(* Logix 5000 project; controller Sucrose_Main Emulate 5570 rev 20.12; software revision 20.01; part 12 of 30 *)
(* tags used below, declared in another part *)
   AI_E21_0 : REAL[8];   // Analog Input EN2T_FLX 192.168.1.21
   AI_E21_1 : REAL[8];   // Analog Input EN2T_FLX 192.168.1.21
   AI_E21_2 : REAL[8];   // Analog Input EN2T_FLX 192.168.1.21
   HOT_WATER_FLOW : DINT;
   HOT_WATER_TEMP : DINT;
   HRM_SIP250TimeRemaining : DINT;
   HRM_SIP254TimeRemaining : DINT;
   HRM_StepTimeRemaining : DINT;
   Integrity_Control : CONTROL;
   Integrity_Result : DINT;
   Integrity_Test_FIFO : REAL[15];
   New_Sec : BOOL;
   ONESHOTBITS : INT[10];
   Rung_Comment : BOOL;
   SucroseDischarge : Area_Program;
   SucroseFiltration : Area_Program;
   temp_toggle : BOOL;
   toggle : BOOL;
(* FiltrationArea_AutoLogic, continued *)

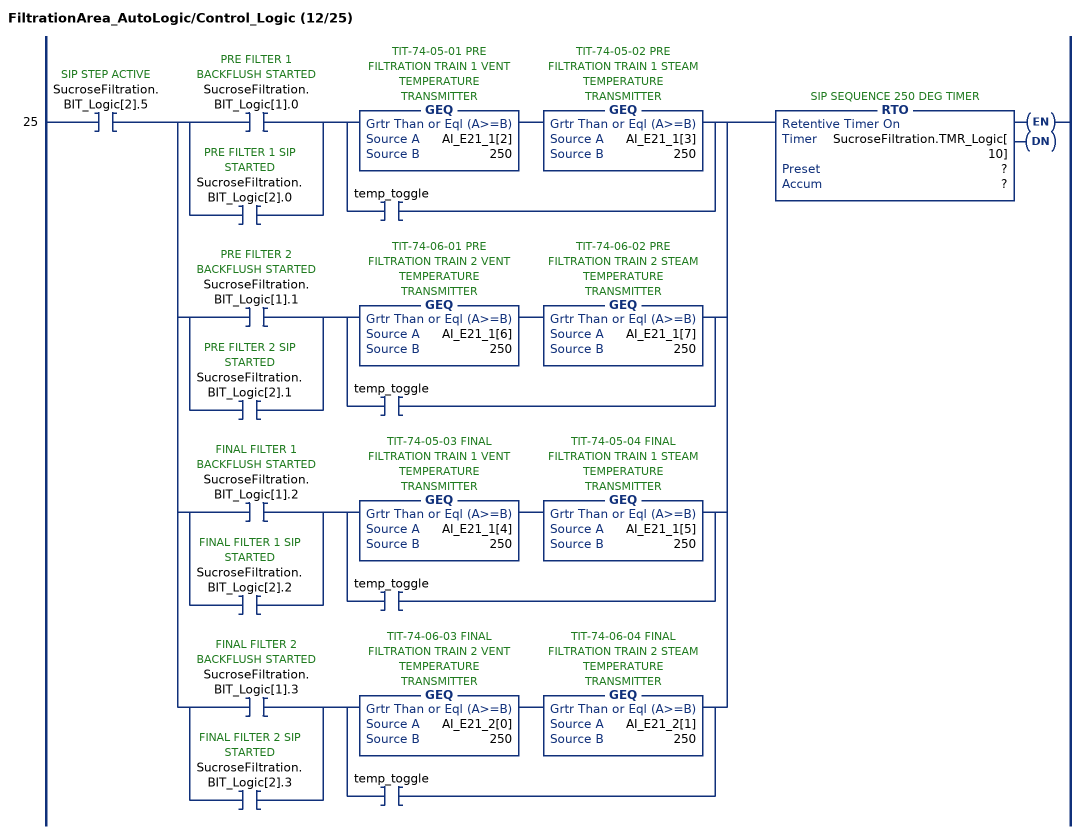
   25: XIC(SucroseFiltration.BIT_Logic[2].5)[[XIC(SucroseFiltration.BIT_Logic[1].0) ,XIC(SucroseFiltration.BIT_Logic[2].0) ] [GEQ(AI_E21_1[2],250) GEQ(AI_E21_1[3],250) ,XIC(temp_toggle) ] ,[XIC(SucroseFiltration.BIT_Logic[1].1) ,XIC(SucroseFiltration.BIT_Logic[2].1) ] [GEQ(AI_E21_1[6],250) GEQ(AI_E21_1[7],250) ,XIC(temp_toggle) ] ,[XIC(SucroseFiltration.BIT_Logic[1].2) ,XIC(SucroseFiltration.BIT_Logic[2].2) ] [GEQ(AI_E21_1[4],250) GEQ(AI_E21_1[5],250) ,XIC(temp_toggle) ] ,[XIC(SucroseFiltration.BIT_Logic[1].3) ,XIC(SucroseFiltration.BIT_Logic[2].3) ] [GEQ(AI_E21_2[0],250) GEQ(AI_E21_2[1],250) ,XIC(temp_toggle) ] ]RTO(SucroseFiltration.TMR_Logic[10],?,?);
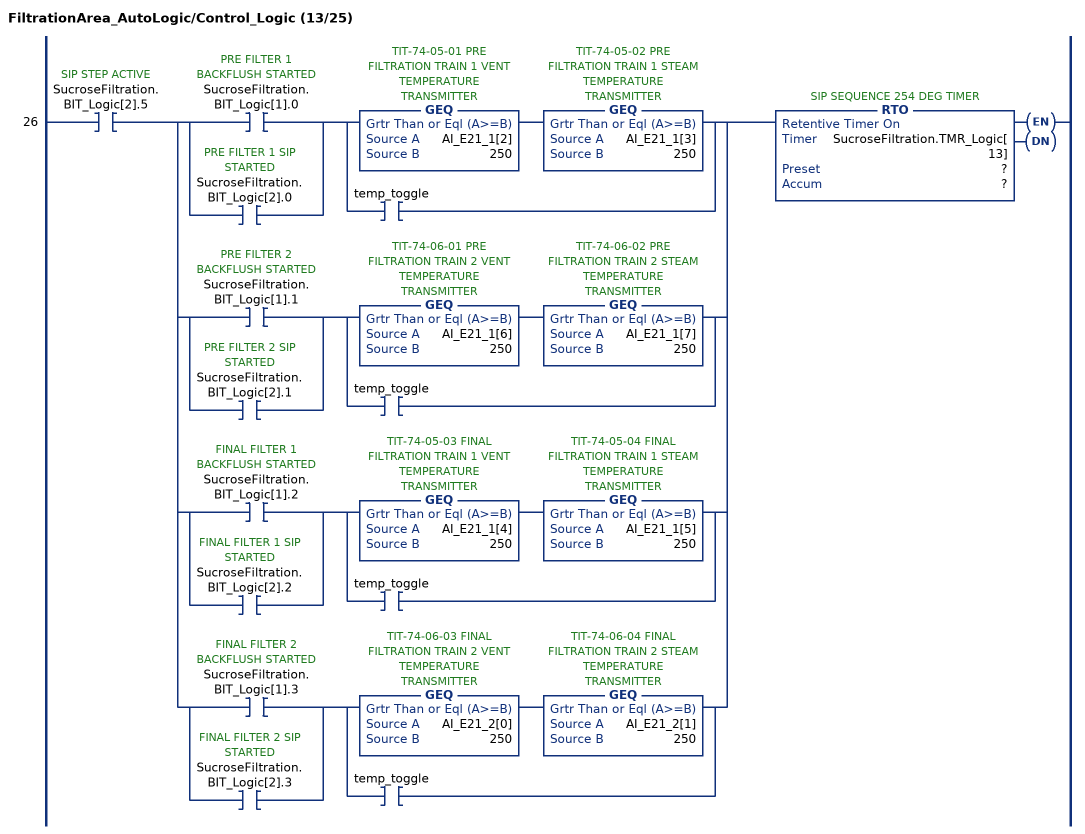
   26: XIC(SucroseFiltration.BIT_Logic[2].5)[[XIC(SucroseFiltration.BIT_Logic[1].0) ,XIC(SucroseFiltration.BIT_Logic[2].0) ] [GEQ(AI_E21_1[2],250) GEQ(AI_E21_1[3],250) ,XIC(temp_toggle) ] ,[XIC(SucroseFiltration.BIT_Logic[1].1) ,XIC(SucroseFiltration.BIT_Logic[2].1) ] [GEQ(AI_E21_1[6],250) GEQ(AI_E21_1[7],250) ,XIC(temp_toggle) ] ,[XIC(SucroseFiltration.BIT_Logic[1].2) ,XIC(SucroseFiltration.BIT_Logic[2].2) ] [GEQ(AI_E21_1[4],250) GEQ(AI_E21_1[5],250) ,XIC(temp_toggle) ] ,[XIC(SucroseFiltration.BIT_Logic[1].3) ,XIC(SucroseFiltration.BIT_Logic[2].3) ] [GEQ(AI_E21_2[0],250) GEQ(AI_E21_2[1],250) ,XIC(temp_toggle) ] ]RTO(SucroseFiltration.TMR_Logic[13],?,?);
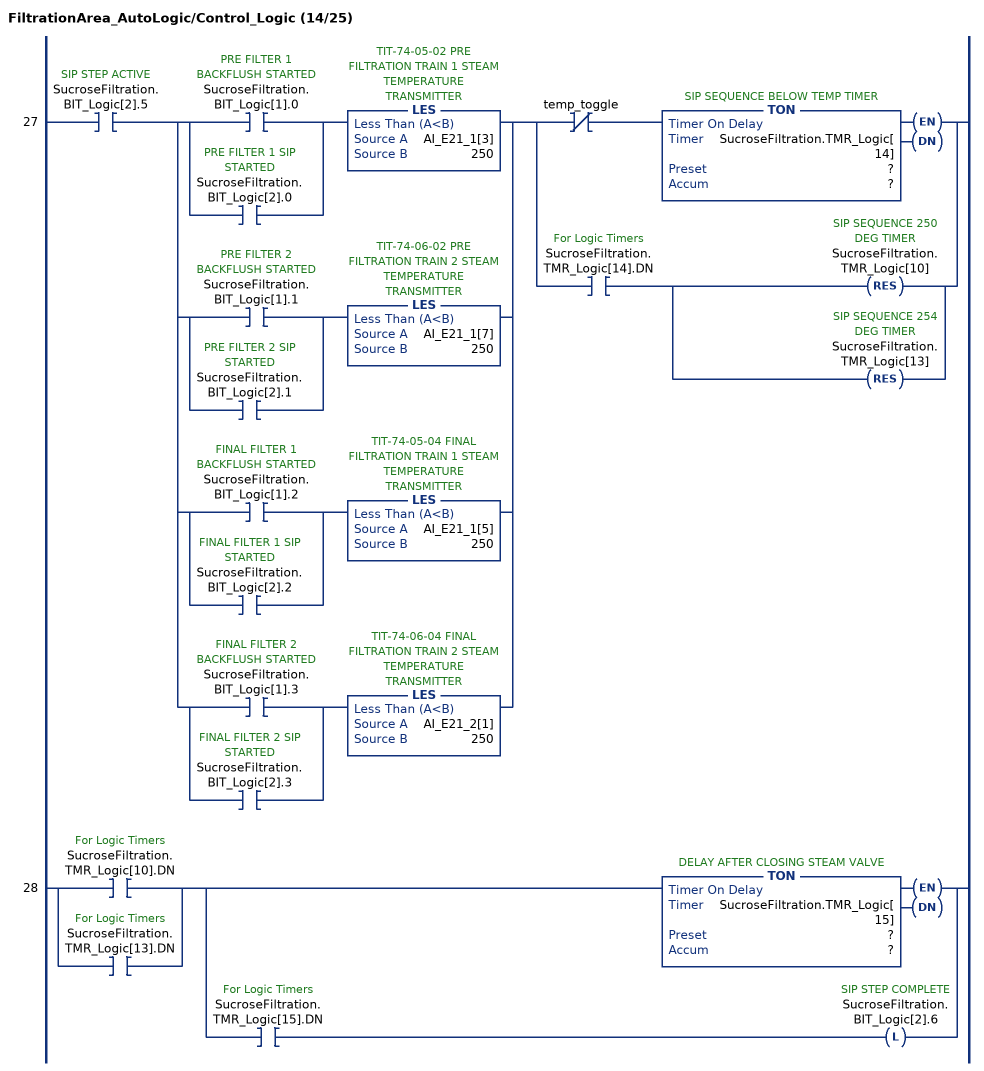
   27: XIC(SucroseFiltration.BIT_Logic[2].5)[[XIC(SucroseFiltration.BIT_Logic[1].0) ,XIC(SucroseFiltration.BIT_Logic[2].0) ] LES(AI_E21_1[3],250) ,[XIC(SucroseFiltration.BIT_Logic[1].1) ,XIC(SucroseFiltration.BIT_Logic[2].1) ] LES(AI_E21_1[7],250) ,[XIC(SucroseFiltration.BIT_Logic[1].2) ,XIC(SucroseFiltration.BIT_Logic[2].2) ] LES(AI_E21_1[5],250) ,[XIC(SucroseFiltration.BIT_Logic[1].3) ,XIC(SucroseFiltration.BIT_Logic[2].3) ] LES(AI_E21_2[1],250) ][XIO(temp_toggle) TON(SucroseFiltration.TMR_Logic[14],?,?) ,XIC(SucroseFiltration.TMR_Logic[14].DN) [RES(SucroseFiltration.TMR_Logic[10]) ,RES(SucroseFiltration.TMR_Logic[13]) ] ];
   28: [XIC(SucroseFiltration.TMR_Logic[10].DN) ,XIC(SucroseFiltration.TMR_Logic[13].DN) ][TON(SucroseFiltration.TMR_Logic[15],?,?) ,XIC(SucroseFiltration.TMR_Logic[15].DN) OTL(SucroseFiltration.BIT_Logic[2].6) ];
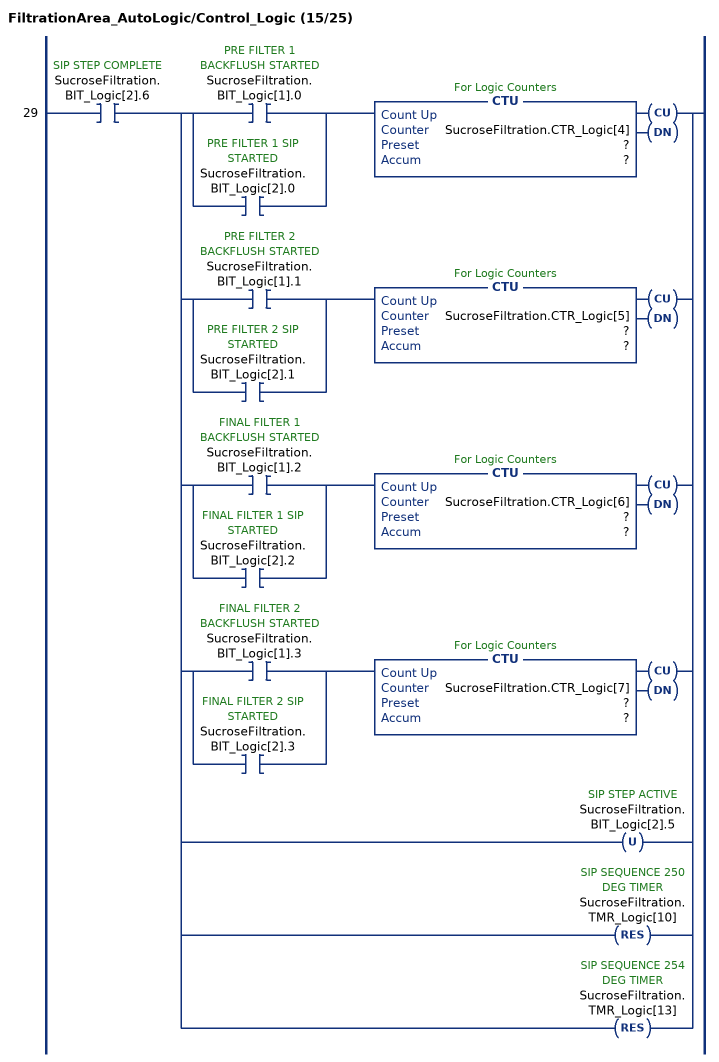
   29: XIC(SucroseFiltration.BIT_Logic[2].6)[[XIC(SucroseFiltration.BIT_Logic[1].0) ,XIC(SucroseFiltration.BIT_Logic[2].0) ] CTU(SucroseFiltration.CTR_Logic[4],?,?) ,[XIC(SucroseFiltration.BIT_Logic[1].1) ,XIC(SucroseFiltration.BIT_Logic[2].1) ] CTU(SucroseFiltration.CTR_Logic[5],?,?) ,[XIC(SucroseFiltration.BIT_Logic[1].2) ,XIC(SucroseFiltration.BIT_Logic[2].2) ] CTU(SucroseFiltration.CTR_Logic[6],?,?) ,[XIC(SucroseFiltration.BIT_Logic[1].3) ,XIC(SucroseFiltration.BIT_Logic[2].3) ] CTU(SucroseFiltration.CTR_Logic[7],?,?) ,OTU(SucroseFiltration.BIT_Logic[2].5) ,RES(SucroseFiltration.TMR_Logic[10]) ,RES(SucroseFiltration.TMR_Logic[13]) ];
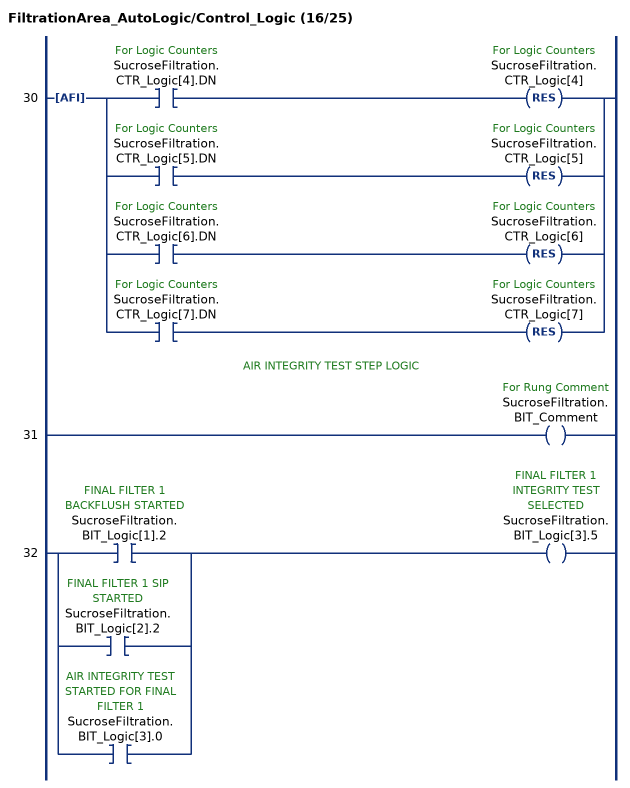
   30: AFI()[XIC(SucroseFiltration.CTR_Logic[4].DN) RES(SucroseFiltration.CTR_Logic[4]) ,XIC(SucroseFiltration.CTR_Logic[5].DN) RES(SucroseFiltration.CTR_Logic[5]) ,XIC(SucroseFiltration.CTR_Logic[6].DN) RES(SucroseFiltration.CTR_Logic[6]) ,XIC(SucroseFiltration.CTR_Logic[7].DN) RES(SucroseFiltration.CTR_Logic[7]) ];
   // AIR INTEGRITY TEST STEP LOGIC
   31: OTE(SucroseFiltration.BIT_Comment);
   32: [XIC(SucroseFiltration.BIT_Logic[1].2) ,XIC(SucroseFiltration.BIT_Logic[2].2) ,XIC(SucroseFiltration.BIT_Logic[3].0) ]OTE(SucroseFiltration.BIT_Logic[3].5);
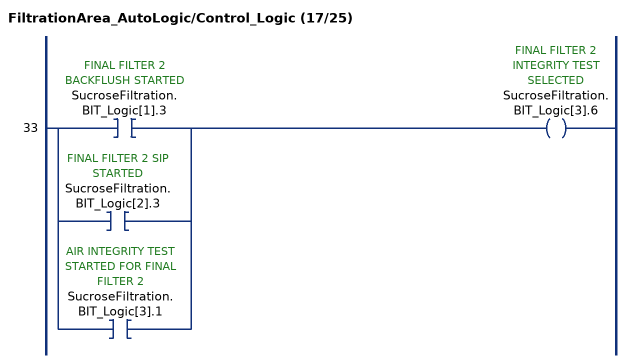
   33: [XIC(SucroseFiltration.BIT_Logic[1].3) ,XIC(SucroseFiltration.BIT_Logic[2].3) ,XIC(SucroseFiltration.BIT_Logic[3].1) ]OTE(SucroseFiltration.BIT_Logic[3].6);
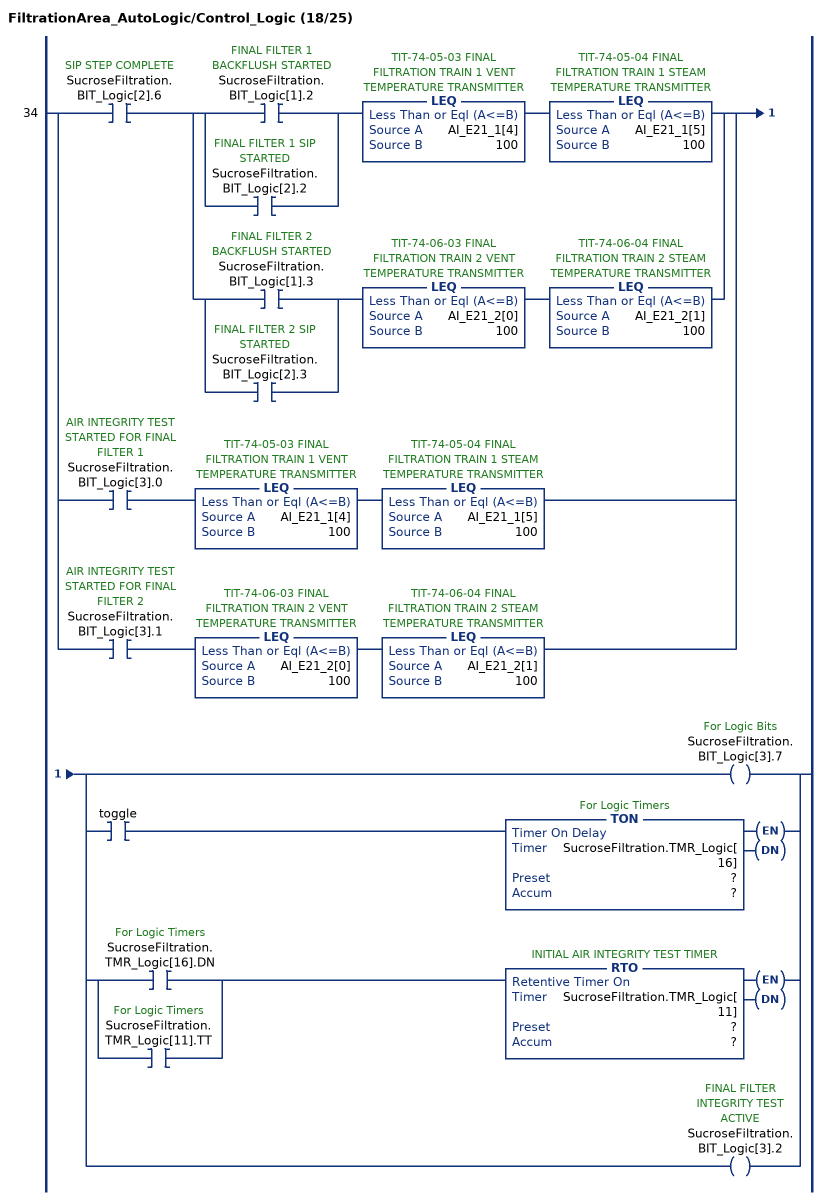
   34: [XIC(SucroseFiltration.BIT_Logic[2].6) [[XIC(SucroseFiltration.BIT_Logic[1].2) ,XIC(SucroseFiltration.BIT_Logic[2].2) ] LEQ(AI_E21_1[4],100) LEQ(AI_E21_1[5],100) ,[XIC(SucroseFiltration.BIT_Logic[1].3) ,XIC(SucroseFiltration.BIT_Logic[2].3) ] LEQ(AI_E21_2[0],100) LEQ(AI_E21_2[1],100) ] ,[XIC(SucroseFiltration.BIT_Logic[3].0) LEQ(AI_E21_1[4],100) LEQ(AI_E21_1[5],100) ,XIC(SucroseFiltration.BIT_Logic[3].1) LEQ(AI_E21_2[0],100) LEQ(AI_E21_2[1],100) ] ][OTE(SucroseFiltration.BIT_Logic[3].7) ,XIC(toggle) TON(SucroseFiltration.TMR_Logic[16],?,?) ,[XIC(SucroseFiltration.TMR_Logic[16].DN) ,XIC(SucroseFiltration.TMR_Logic[11].TT) ] RTO(SucroseFiltration.TMR_Logic[11],?,?) ,OTE(SucroseFiltration.BIT_Logic[3].2) ];
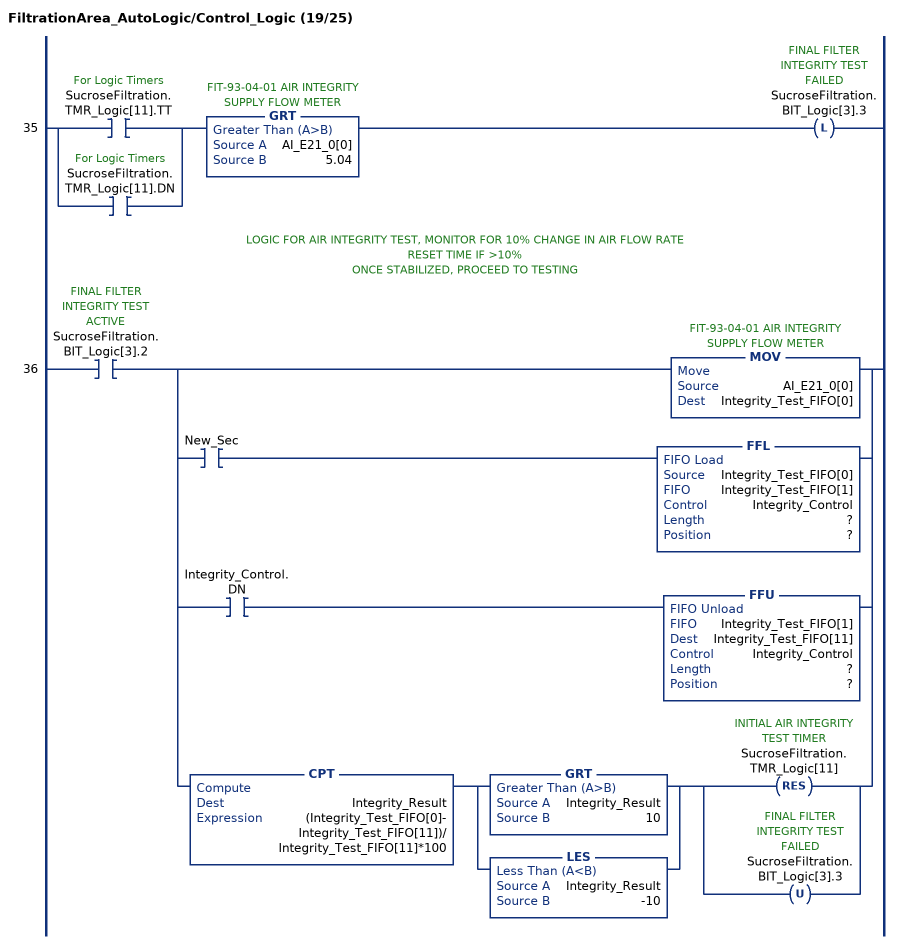
   35: [XIC(SucroseFiltration.TMR_Logic[11].TT) ,XIC(SucroseFiltration.TMR_Logic[11].DN) ]GRT(AI_E21_0[0],5.04)OTL(SucroseFiltration.BIT_Logic[3].3);
   // LOGIC FOR AIR INTEGRITY TEST, MONITOR FOR 10% CHANGE IN AIR FLOW RATE
   // RESET TIME IF >10%
   // ONCE STABILIZED, PROCEED TO TESTING
   36: XIC(SucroseFiltration.BIT_Logic[3].2)[MOV(AI_E21_0[0],Integrity_Test_FIFO[0]) ,XIC(New_Sec) FFL(Integrity_Test_FIFO[0],Integrity_Test_FIFO[1],Integrity_Control,?,?) ,XIC(Integrity_Control.DN) FFU(Integrity_Test_FIFO[1],Integrity_Test_FIFO[11],Integrity_Control,?,?) ,CPT(Integrity_Result,(Integrity_Test_FIFO[0]-Integrity_Test_FIFO[11])/Integrity_Test_FIFO[11]*100) [GRT(Integrity_Result,10) ,LES(Integrity_Result,-10) ] [RES(SucroseFiltration.TMR_Logic[11]) ,OTU(SucroseFiltration.BIT_Logic[3].3) ] ];
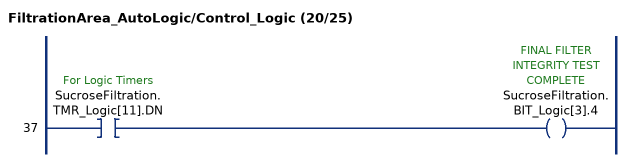
   37: XIC(SucroseFiltration.TMR_Logic[11].DN)OTE(SucroseFiltration.BIT_Logic[3].4);
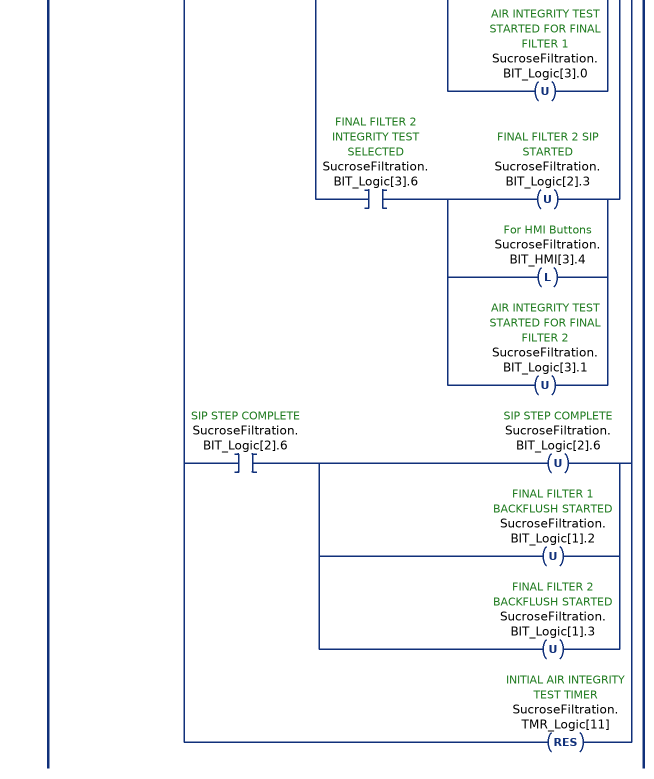
   38: XIC(SucroseFiltration.TMR_Logic[11].DN)[XIO(SucroseFiltration.BIT_Logic[3].3) [XIC(SucroseFiltration.BIT_Logic[3].5) [OTL(SucroseFiltration.BIT_Logic[0].3) ,OTU(SucroseFiltration.BIT_Logic[2].2) ,OTU(SucroseFiltration.BIT_Logic[3].0) ,OTU(SucroseFiltration.BIT_HMI[3].3) ] ,XIC(SucroseFiltration.BIT_Logic[3].6) [OTL(SucroseFiltration.BIT_Logic[0].4) ,OTU(SucroseFiltration.BIT_Logic[2].3) ,OTU(SucroseFiltration.BIT_Logic[3].1) ,OTU(SucroseFiltration.BIT_HMI[3].4) ] ] ,XIC(SucroseFiltration.BIT_Logic[3].3) [XIC(SucroseFiltration.BIT_Logic[3].5) [OTU(SucroseFiltration.BIT_Logic[2].2) ,OTL(SucroseFiltration.BIT_HMI[3].3) ,OTU(SucroseFiltration.BIT_Logic[3].0) ] ,XIC(SucroseFiltration.BIT_Logic[3].6) [OTU(SucroseFiltration.BIT_Logic[2].3) ,OTL(SucroseFiltration.BIT_HMI[3].4) ,OTU(SucroseFiltration.BIT_Logic[3].1) ] ] ,XIC(SucroseFiltration.BIT_Logic[2].6) [OTU(SucroseFiltration.BIT_Logic[2].6) ,OTU(SucroseFiltration.BIT_Logic[1].2) ,OTU(SucroseFiltration.BIT_Logic[1].3) ] ,RES(SucroseFiltration.TMR_Logic[11]) ];
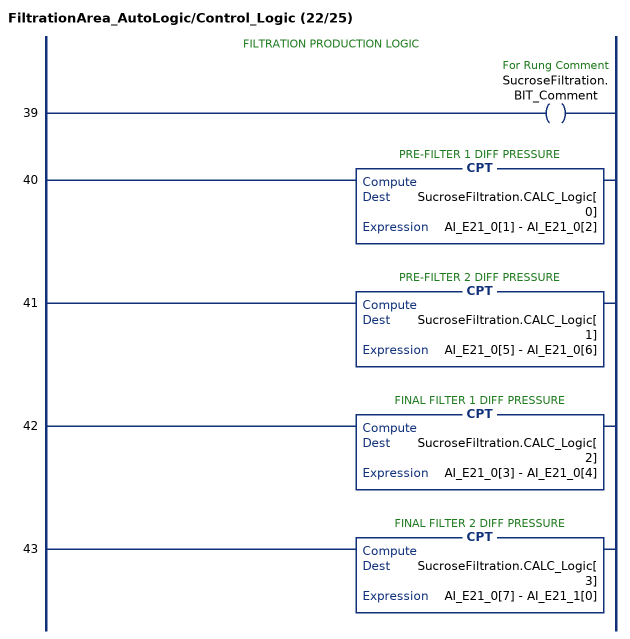
   // FILTRATION PRODUCTION LOGIC
   39: OTE(SucroseFiltration.BIT_Comment);
   40: CPT(SucroseFiltration.CALC_Logic[0],AI_E21_0[1] - AI_E21_0[2]);
   41: CPT(SucroseFiltration.CALC_Logic[1],AI_E21_0[5] - AI_E21_0[6]);
   42: CPT(SucroseFiltration.CALC_Logic[2],AI_E21_0[3] - AI_E21_0[4]);
   43: CPT(SucroseFiltration.CALC_Logic[3],AI_E21_0[7] - AI_E21_1[0]);
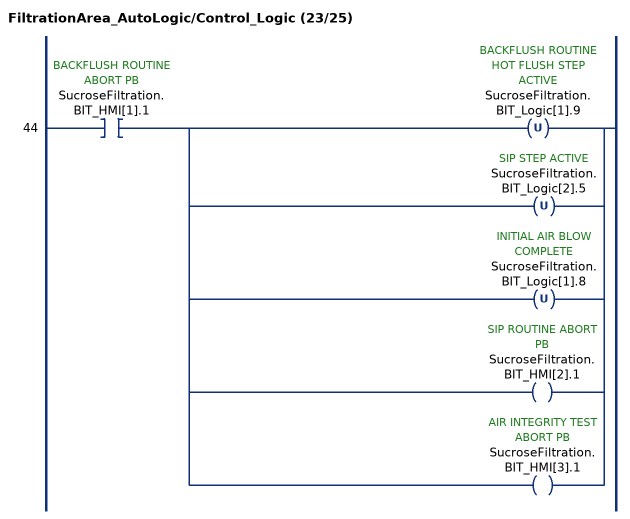
   44: XIC(SucroseFiltration.BIT_HMI[1].1)[OTU(SucroseFiltration.BIT_Logic[1].9) ,OTU(SucroseFiltration.BIT_Logic[2].5) ,OTU(SucroseFiltration.BIT_Logic[1].8) ,OTE(SucroseFiltration.BIT_HMI[2].1) ,OTE(SucroseFiltration.BIT_HMI[3].1) ];
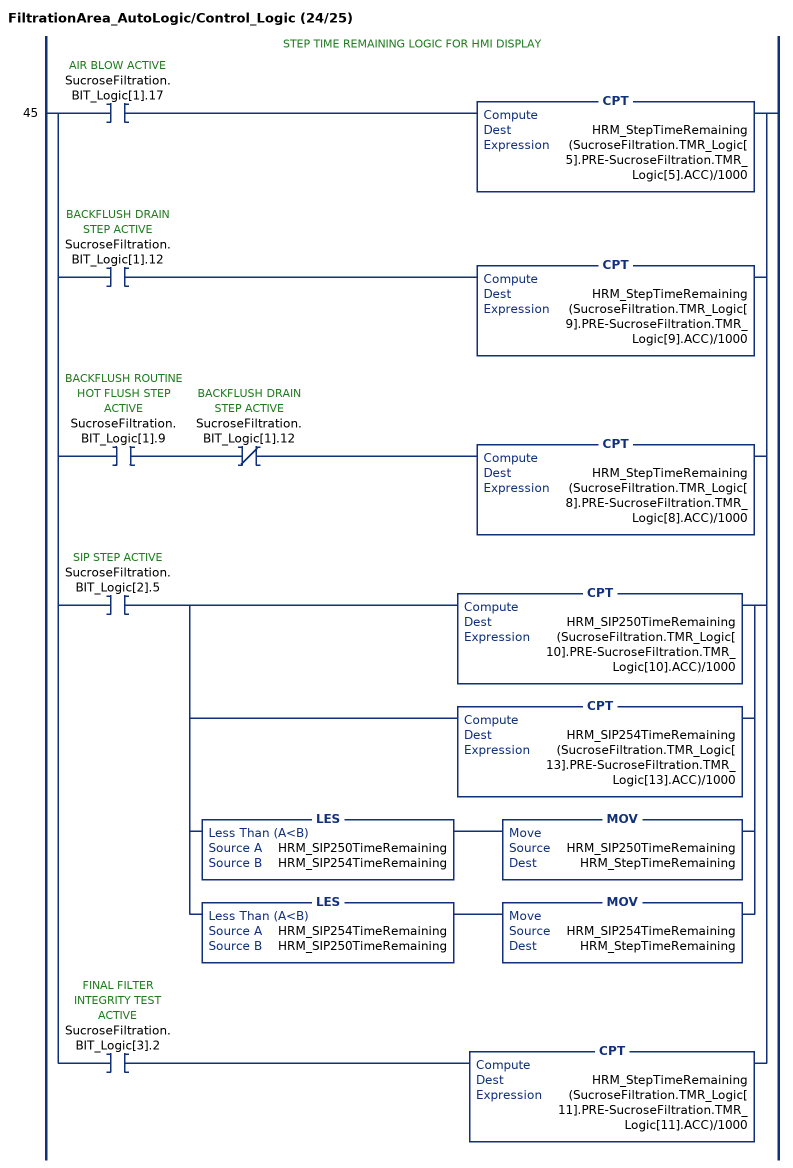
   // STEP TIME REMAINING LOGIC FOR HMI DISPLAY
   45: [XIC(SucroseFiltration.BIT_Logic[1].17) CPT(HRM_StepTimeRemaining,(SucroseFiltration.TMR_Logic[5].PRE-SucroseFiltration.TMR_Logic[5].ACC)/1000) ,XIC(SucroseFiltration.BIT_Logic[1].12) CPT(HRM_StepTimeRemaining,(SucroseFiltration.TMR_Logic[9].PRE-SucroseFiltration.TMR_Logic[9].ACC)/1000) ,XIC(SucroseFiltration.BIT_Logic[1].9) XIO(SucroseFiltration.BIT_Logic[1].12) CPT(HRM_StepTimeRemaining,(SucroseFiltration.TMR_Logic[8].PRE-SucroseFiltration.TMR_Logic[8].ACC)/1000) ,XIC(SucroseFiltration.BIT_Logic[2].5) [CPT(HRM_SIP250TimeRemaining,(SucroseFiltration.TMR_Logic[10].PRE-SucroseFiltration.TMR_Logic[10].ACC)/1000) ,CPT(HRM_SIP254TimeRemaining,(SucroseFiltration.TMR_Logic[13].PRE-SucroseFiltration.TMR_Logic[13].ACC)/1000) ,LES(HRM_SIP250TimeRemaining,HRM_SIP254TimeRemaining) MOV(HRM_SIP250TimeRemaining,HRM_StepTimeRemaining) ,LES(HRM_SIP254TimeRemaining,HRM_SIP250TimeRemaining) MOV(HRM_SIP254TimeRemaining,HRM_StepTimeRemaining) ] ,XIC(SucroseFiltration.BIT_Logic[3].2) CPT(HRM_StepTimeRemaining,(SucroseFiltration.TMR_Logic[11].PRE-SucroseFiltration.TMR_Logic[11].ACC)/1000) ];
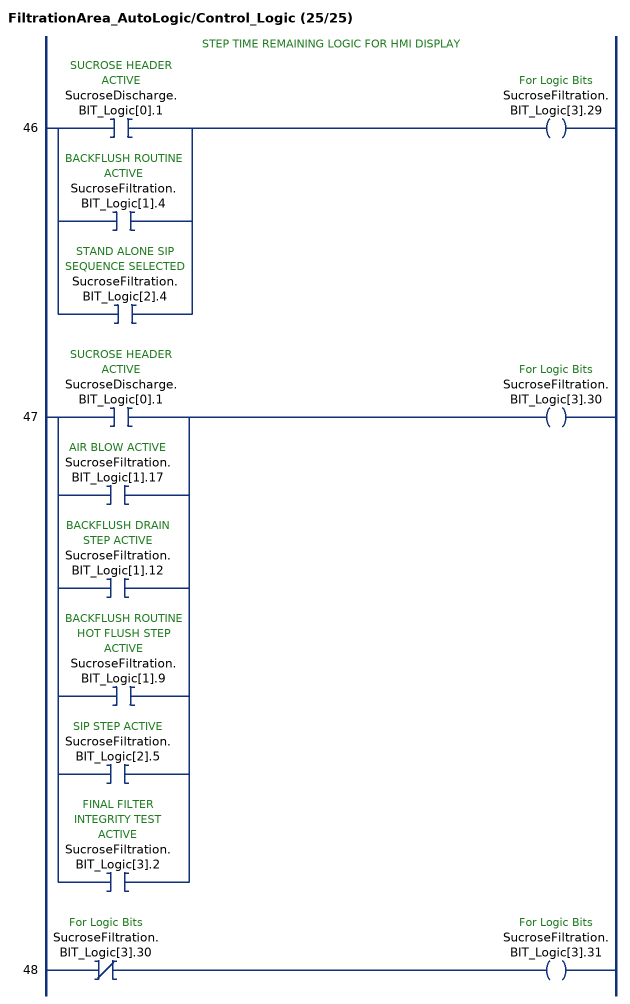
   // STEP TIME REMAINING LOGIC FOR HMI DISPLAY
   46: [XIC(SucroseDischarge.BIT_Logic[0].1) ,XIC(SucroseFiltration.BIT_Logic[1].4) ,XIC(SucroseFiltration.BIT_Logic[2].4) ]OTE(SucroseFiltration.BIT_Logic[3].29);
   47: [XIC(SucroseDischarge.BIT_Logic[0].1) ,XIC(SucroseFiltration.BIT_Logic[1].17) ,XIC(SucroseFiltration.BIT_Logic[1].12) ,XIC(SucroseFiltration.BIT_Logic[1].9) ,XIC(SucroseFiltration.BIT_Logic[2].5) ,XIC(SucroseFiltration.BIT_Logic[3].2) ]OTE(SucroseFiltration.BIT_Logic[3].30);
   48: XIO(SucroseFiltration.BIT_Logic[3].30)OTE(SucroseFiltration.BIT_Logic[3].31);
END_ROUTINE

ROUTINE Control_Logic_old   (* ladder *)
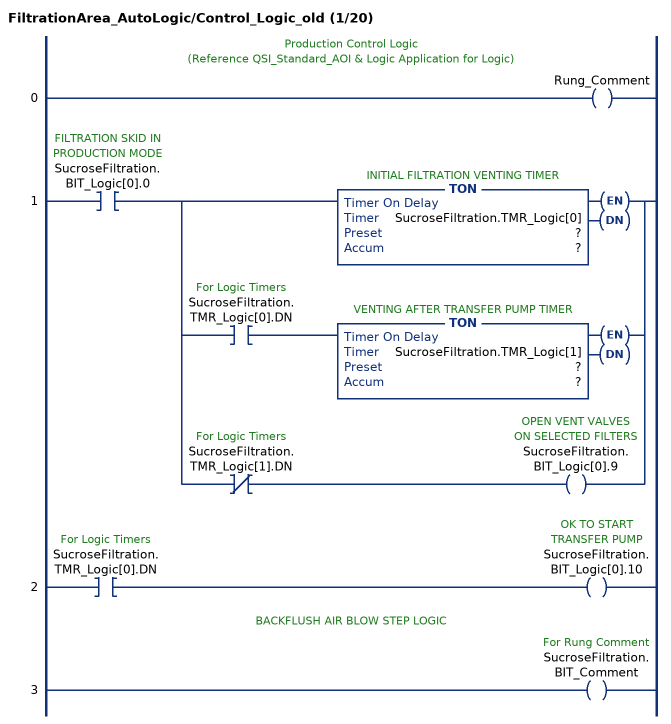
   // Production Control Logic
   // (Reference QSI_Standard_AOI & Logic Application for Logic)
   0: OTE(Rung_Comment);
   1: XIC(SucroseFiltration.BIT_Logic[0].0)[TON(SucroseFiltration.TMR_Logic[0],?,?) ,XIC(SucroseFiltration.TMR_Logic[0].DN) TON(SucroseFiltration.TMR_Logic[1],?,?) ,XIO(SucroseFiltration.TMR_Logic[1].DN) OTE(SucroseFiltration.BIT_Logic[0].9) ];
   2: XIC(SucroseFiltration.TMR_Logic[0].DN)OTE(SucroseFiltration.BIT_Logic[0].10);
   // BACKFLUSH AIR BLOW STEP LOGIC
   3: OTE(SucroseFiltration.BIT_Comment);
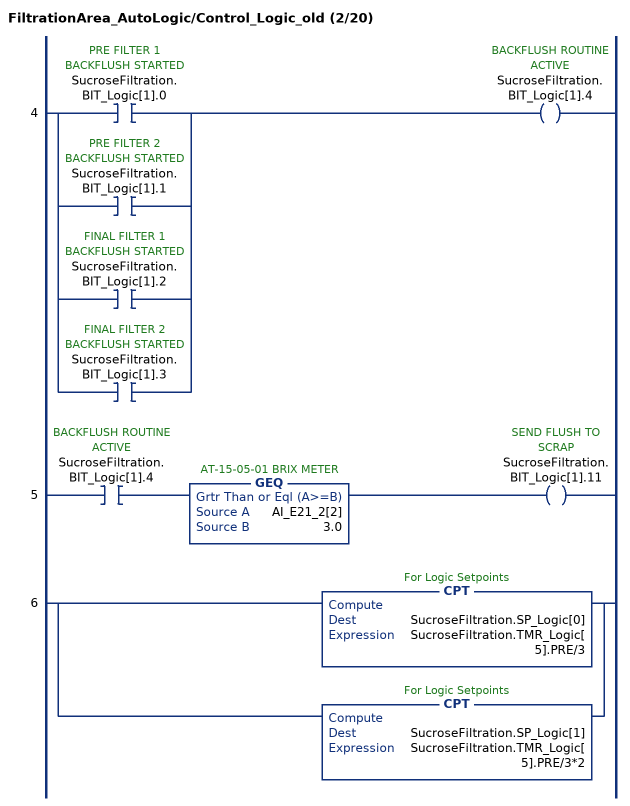
   4: [XIC(SucroseFiltration.BIT_Logic[1].0) ,XIC(SucroseFiltration.BIT_Logic[1].1) ,XIC(SucroseFiltration.BIT_Logic[1].2) ,XIC(SucroseFiltration.BIT_Logic[1].3) ]OTE(SucroseFiltration.BIT_Logic[1].4);
   5: XIC(SucroseFiltration.BIT_Logic[1].4)GEQ(AI_E21_2[2],3.0)OTE(SucroseFiltration.BIT_Logic[1].11);
   6: [CPT(SucroseFiltration.SP_Logic[0],SucroseFiltration.TMR_Logic[5].PRE/3) ,CPT(SucroseFiltration.SP_Logic[1],SucroseFiltration.TMR_Logic[5].PRE/3*2) ];
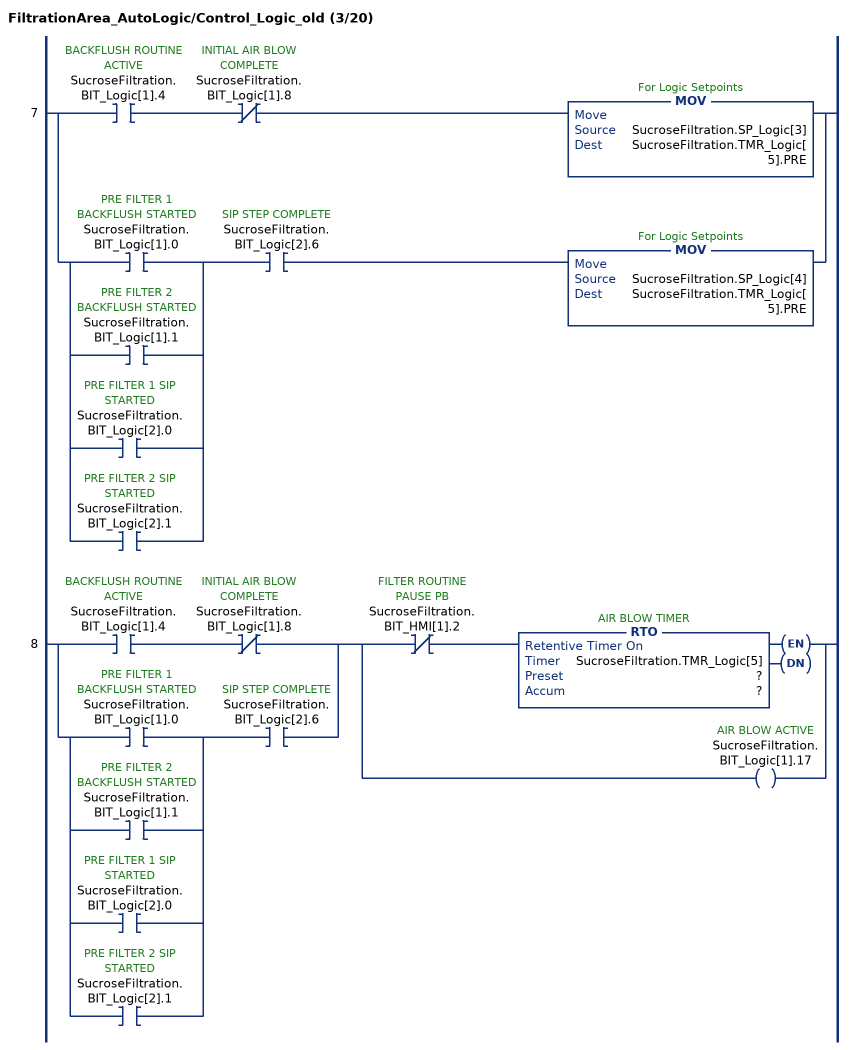
   7: [XIC(SucroseFiltration.BIT_Logic[1].4) XIO(SucroseFiltration.BIT_Logic[1].8) MOV(SucroseFiltration.SP_Logic[3],SucroseFiltration.TMR_Logic[5].PRE) ,[XIC(SucroseFiltration.BIT_Logic[1].0) ,XIC(SucroseFiltration.BIT_Logic[1].1) ,XIC(SucroseFiltration.BIT_Logic[2].0) ,XIC(SucroseFiltration.BIT_Logic[2].1) ] XIC(SucroseFiltration.BIT_Logic[2].6) MOV(SucroseFiltration.SP_Logic[4],SucroseFiltration.TMR_Logic[5].PRE) ];
   8: [XIC(SucroseFiltration.BIT_Logic[1].4) XIO(SucroseFiltration.BIT_Logic[1].8) ,[XIC(SucroseFiltration.BIT_Logic[1].0) ,XIC(SucroseFiltration.BIT_Logic[1].1) ,XIC(SucroseFiltration.BIT_Logic[2].0) ,XIC(SucroseFiltration.BIT_Logic[2].1) ] XIC(SucroseFiltration.BIT_Logic[2].6) ][XIO(SucroseFiltration.BIT_HMI[1].2) RTO(SucroseFiltration.TMR_Logic[5],?,?) ,OTE(SucroseFiltration.BIT_Logic[1].17) ];
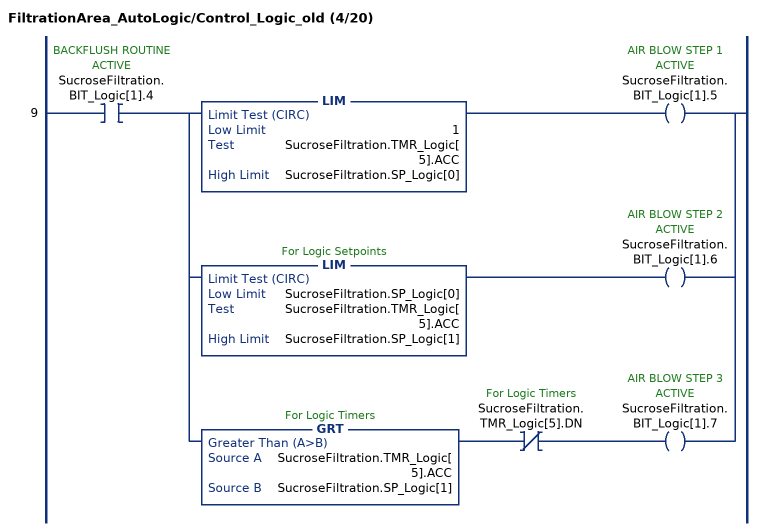
   9: XIC(SucroseFiltration.BIT_Logic[1].4)[LIM(1,SucroseFiltration.TMR_Logic[5].ACC,SucroseFiltration.SP_Logic[0]) OTE(SucroseFiltration.BIT_Logic[1].5) ,LIM(SucroseFiltration.SP_Logic[0],SucroseFiltration.TMR_Logic[5].ACC,SucroseFiltration.SP_Logic[1]) OTE(SucroseFiltration.BIT_Logic[1].6) ,GRT(SucroseFiltration.TMR_Logic[5].ACC,SucroseFiltration.SP_Logic[1]) XIO(SucroseFiltration.TMR_Logic[5].DN) OTE(SucroseFiltration.BIT_Logic[1].7) ];
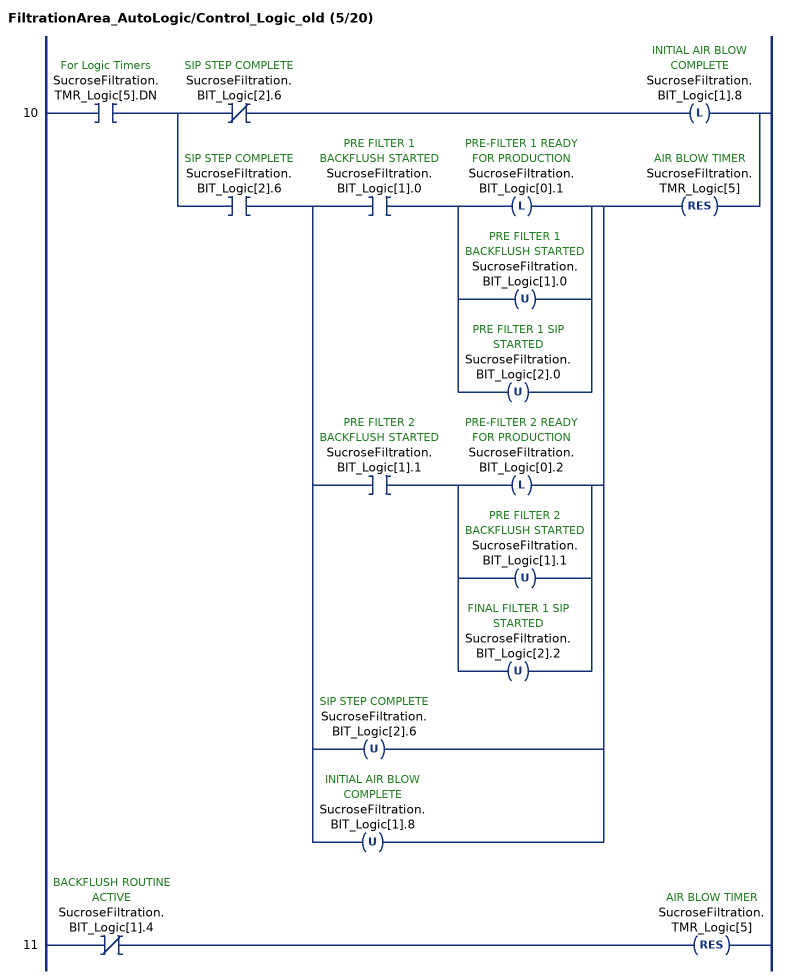
   10: XIC(SucroseFiltration.TMR_Logic[5].DN)[XIO(SucroseFiltration.BIT_Logic[2].6) OTL(SucroseFiltration.BIT_Logic[1].8) ,XIC(SucroseFiltration.BIT_Logic[2].6) [XIC(SucroseFiltration.BIT_Logic[1].0) [OTL(SucroseFiltration.BIT_Logic[0].1) ,OTU(SucroseFiltration.BIT_Logic[1].0) ,OTU(SucroseFiltration.BIT_Logic[2].0) ] ,XIC(SucroseFiltration.BIT_Logic[1].1) [OTL(SucroseFiltration.BIT_Logic[0].2) ,OTU(SucroseFiltration.BIT_Logic[1].1) ,OTU(SucroseFiltration.BIT_Logic[2].2) ] ,OTU(SucroseFiltration.BIT_Logic[2].6) ,OTU(SucroseFiltration.BIT_Logic[1].8) ] RES(SucroseFiltration.TMR_Logic[5]) ];
   11: XIO(SucroseFiltration.BIT_Logic[1].4)RES(SucroseFiltration.TMR_Logic[5]);
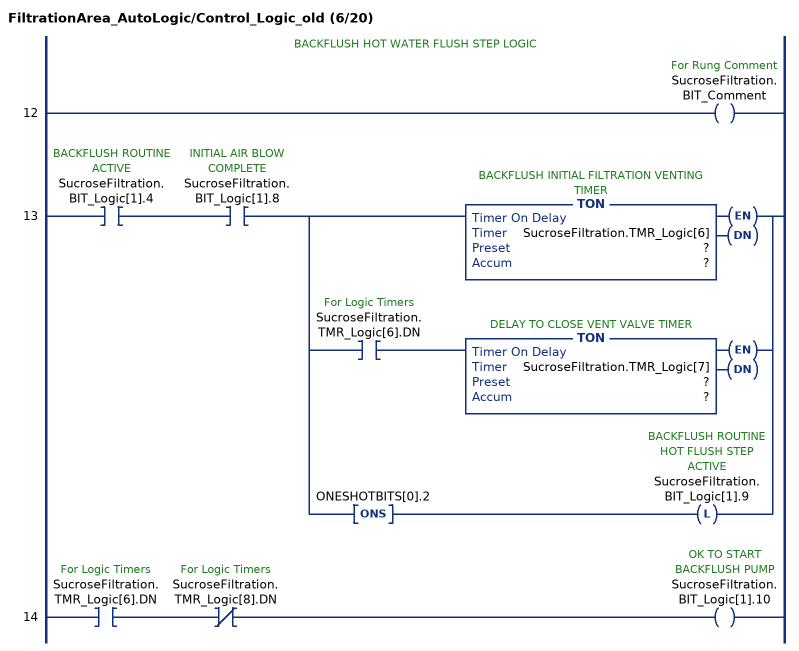
   // BACKFLUSH HOT WATER FLUSH STEP LOGIC
   12: OTE(SucroseFiltration.BIT_Comment);
   13: XIC(SucroseFiltration.BIT_Logic[1].4)XIC(SucroseFiltration.BIT_Logic[1].8)[TON(SucroseFiltration.TMR_Logic[6],?,?) ,XIC(SucroseFiltration.TMR_Logic[6].DN) TON(SucroseFiltration.TMR_Logic[7],?,?) ,ONS(ONESHOTBITS[0].2) OTL(SucroseFiltration.BIT_Logic[1].9) ];
   14: XIC(SucroseFiltration.TMR_Logic[6].DN)XIO(SucroseFiltration.TMR_Logic[8].DN)OTE(SucroseFiltration.BIT_Logic[1].10);
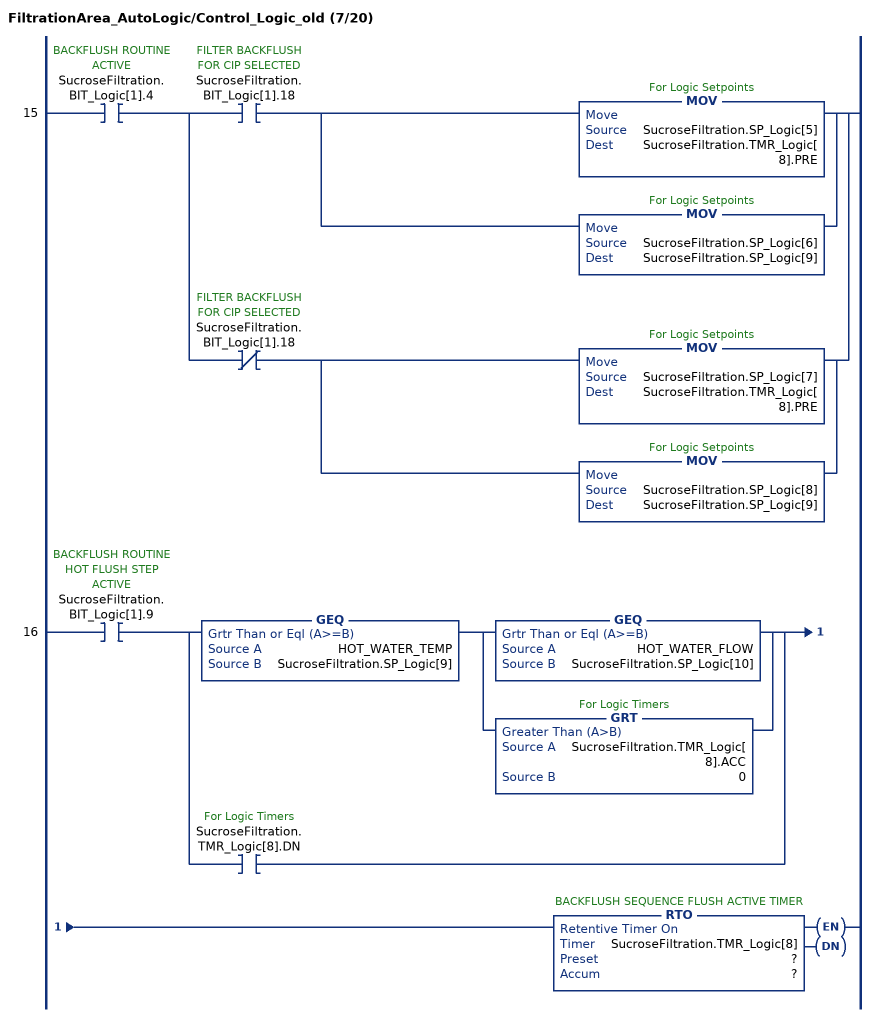
   15: XIC(SucroseFiltration.BIT_Logic[1].4)[XIC(SucroseFiltration.BIT_Logic[1].18) [MOV(SucroseFiltration.SP_Logic[5],SucroseFiltration.TMR_Logic[8].PRE) ,MOV(SucroseFiltration.SP_Logic[6],SucroseFiltration.SP_Logic[9]) ] ,XIO(SucroseFiltration.BIT_Logic[1].18) [MOV(SucroseFiltration.SP_Logic[7],SucroseFiltration.TMR_Logic[8].PRE) ,MOV(SucroseFiltration.SP_Logic[8],SucroseFiltration.SP_Logic[9]) ] ];
   16: XIC(SucroseFiltration.BIT_Logic[1].9)[GEQ(HOT_WATER_TEMP,SucroseFiltration.SP_Logic[9]) [GEQ(HOT_WATER_FLOW,SucroseFiltration.SP_Logic[10]) ,GRT(SucroseFiltration.TMR_Logic[8].ACC,0) ] ,XIC(SucroseFiltration.TMR_Logic[8].DN) ]RTO(SucroseFiltration.TMR_Logic[8],?,?);
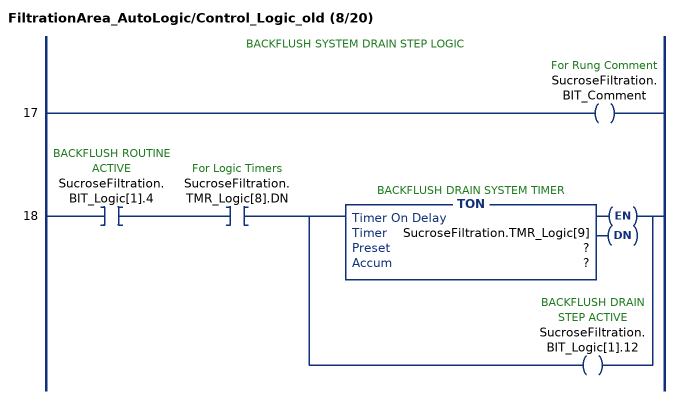
   // BACKFLUSH SYSTEM DRAIN STEP LOGIC
   17: OTE(SucroseFiltration.BIT_Comment);
   18: XIC(SucroseFiltration.BIT_Logic[1].4)XIC(SucroseFiltration.TMR_Logic[8].DN)[TON(SucroseFiltration.TMR_Logic[9],?,?) ,OTE(SucroseFiltration.BIT_Logic[1].12) ];
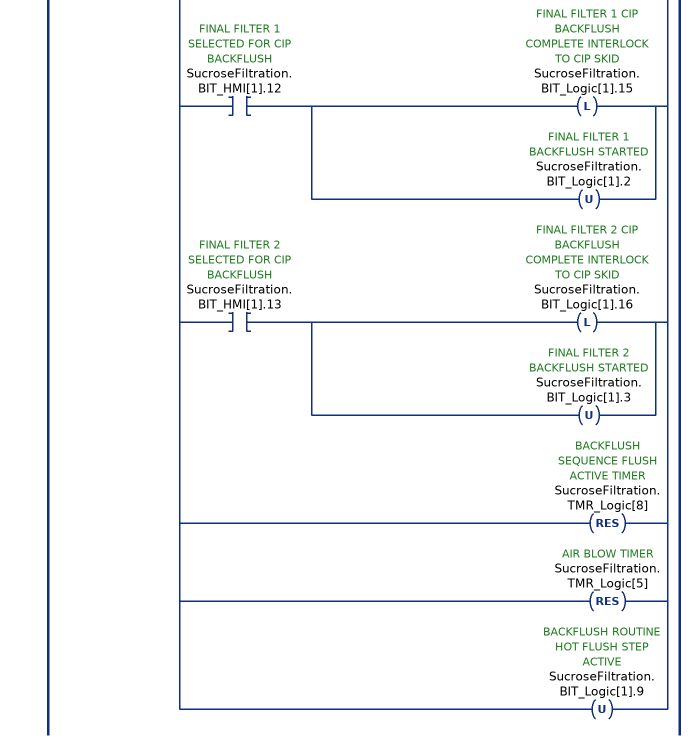
   19: XIC(SucroseFiltration.TMR_Logic[9].DN)[XIC(SucroseFiltration.BIT_Logic[1].0) CTU(SucroseFiltration.CTR_Logic[0],?,?) ,XIC(SucroseFiltration.BIT_Logic[1].1) CTU(SucroseFiltration.CTR_Logic[1],?,?) ,XIC(SucroseFiltration.BIT_Logic[1].2) CTU(SucroseFiltration.CTR_Logic[2],?,?) ,XIC(SucroseFiltration.BIT_Logic[1].3) CTU(SucroseFiltration.CTR_Logic[3],?,?) ,XIC(SucroseFiltration.BIT_HMI[1].10) [OTL(SucroseFiltration.BIT_Logic[1].13) ,OTU(SucroseFiltration.BIT_Logic[1].0) ] ,XIC(SucroseFiltration.BIT_HMI[1].11) [OTL(SucroseFiltration.BIT_Logic[1].14) ,OTU(SucroseFiltration.BIT_Logic[1].1) ] ,XIC(SucroseFiltration.BIT_HMI[1].12) [OTL(SucroseFiltration.BIT_Logic[1].15) ,OTU(SucroseFiltration.BIT_Logic[1].2) ] ,XIC(SucroseFiltration.BIT_HMI[1].13) [OTL(SucroseFiltration.BIT_Logic[1].16) ,OTU(SucroseFiltration.BIT_Logic[1].3) ] ,RES(SucroseFiltration.TMR_Logic[8]) ,RES(SucroseFiltration.TMR_Logic[5]) ,OTU(SucroseFiltration.BIT_Logic[1].9) ];
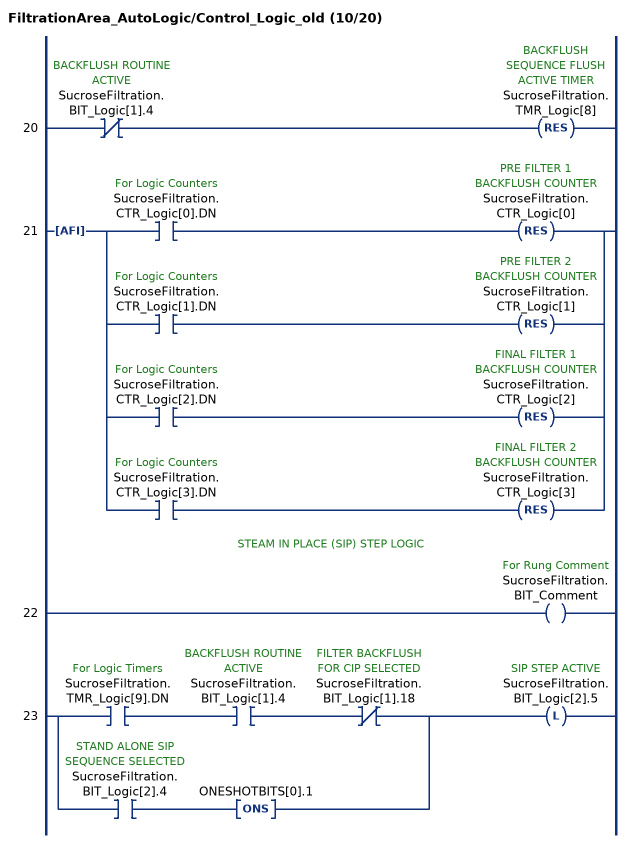
   20: XIO(SucroseFiltration.BIT_Logic[1].4)RES(SucroseFiltration.TMR_Logic[8]);
   21: AFI()[XIC(SucroseFiltration.CTR_Logic[0].DN) RES(SucroseFiltration.CTR_Logic[0]) ,XIC(SucroseFiltration.CTR_Logic[1].DN) RES(SucroseFiltration.CTR_Logic[1]) ,XIC(SucroseFiltration.CTR_Logic[2].DN) RES(SucroseFiltration.CTR_Logic[2]) ,XIC(SucroseFiltration.CTR_Logic[3].DN) RES(SucroseFiltration.CTR_Logic[3]) ];
   // STEAM IN PLACE (SIP) STEP LOGIC
   22: OTE(SucroseFiltration.BIT_Comment);
   23: [XIC(SucroseFiltration.TMR_Logic[9].DN) XIC(SucroseFiltration.BIT_Logic[1].4) XIO(SucroseFiltration.BIT_Logic[1].18) ,XIC(SucroseFiltration.BIT_Logic[2].4) ONS(ONESHOTBITS[0].1) ]OTL(SucroseFiltration.BIT_Logic[2].5);
